{attribute 'GeneratedUsingTerminal: ER8309-1022-0018'}
{attribute addProperty BoxType "ER8309-1022-0018"}
{attribute addProperty Description "ER8309-1022 2Ch. Ana. Input 4-20mA, 1Ch. Pulse Width Current Output (24V, 1.2A), 1 Ch Ana. Output, 2Ch Dig. Out 24V, 0.5A, 4Ch Dig. In. 24V, 4Ch Dig In/Out 24V, 0.5A, M12"}
{attribute addProperty Physics "YY"}
{attribute addProperty Id "AI_Inputs_Channel_1AT %I*AI_Inputs_Channel_A8DF64E310AI_Inputs_Channel_2AT %I*AI_Inputs_Channel_A8DF64E310TACHO_Single_Shaft_Mode_Input_Channel_1AT %I*TACHO_Single_Shaft_Mode_Input_Channel_C331CA3E10DIG_InputsAT %I*DIG_Inputs_495F5DA48PWM_StatusAT %I*PWM_Status_77939B114DEV_InputsAT %I*DEV_Inputs_FBF180A42TACHO_Output_Channel_1AT %Q*TACHO_Output_Channel_600697D91DIG_OutputsAT %Q*DIG_Outputs_0E2843948PWM_ControlAT %Q*PWM_Control_63F162E45WcStateAT %I*WcState_9091E0EB2InfoDataAT %I*InfoData_32EB74EA10"}
{attribute addProperty CRC "2697285495"}
{attribute addProperty Size "70"}
TYPE ER8309_A0C54F77 EXTENDS EtcSlaveBoxBase_77A0E4A7 :
STRUCT
	{attribute addProperty Name "AI_Inputs_Channel_1"}
	AI_Inputs_Channel_1 : AI_Inputs_Channel_A8DF64E3;
	{attribute addProperty Name "AI_Inputs_Channel_2"}
	AI_Inputs_Channel_2 : AI_Inputs_Channel_A8DF64E3;
	{attribute addProperty Name "TACHO_Single_Shaft_Mode_Input_Channel_1"}
	TACHO_Single_Shaft_Mode_Input_Channel_1 : TACHO_Single_Shaft_Mode_Input_Channel_C331CA3E;
	{attribute addProperty Name "DIG_Inputs"}
	DIG_Inputs : DIG_Inputs_495F5DA4;
	{attribute addProperty Name "PWM_Status"}
	PWM_Status : PWM_Status_77939B11;
	{attribute addProperty Name "DEV_Inputs"}
	DEV_Inputs : DEV_Inputs_FBF180A4;
	{attribute addProperty Name "TACHO_Output_Channel_1"}
	TACHO_Output_Channel_1 : TACHO_Output_Channel_600697D9;
	{attribute addProperty Name "DIG_Outputs"}
	DIG_Outputs : DIG_Outputs_0E284394;
	{attribute addProperty Name "PWM_Control"}
	PWM_Control : PWM_Control_63F162E4;
	{attribute addProperty Name "WcState"}
	WcState : WcState_9091E0EB;
	{attribute addProperty Name "InfoData"}
	InfoData : InfoData_32EB74EA;
END_STRUCT
END_TYPE

(* stored: Version 1.2.0.0, ProductVersion 3.1.4024.11
   DUT ER8309_A0C54F77: Id {21e71b6e-c5d2-42dd-ae8d-ba242caf8e00} *)
